(* PLC project 117_1_V0.5.project, CODESYS CODESYS V3.5 SP17 Patch 3 *)
(* stored: creationDateTime 1970-01-01T00:00:00, modificationDateTime 2026-03-26T18:14:32.4070562 *)

FUNCTION_BLOCK TestingForces_150321
  VAR_INPUT
    A : E_A;
  END_VAR
  VAR_OUTPUT
    Fstab : UDINT;
    Fset : UDINT;
    Fsp : UDINT;
    F_su_lower_level : UDINT;
    F_su_upper_level : UDINT;
  END_VAR

            CASE A OF
	
	A60:
				Fstab				:= 50;
				Fset				:= 720;
				Fsp					:= 1575;	
				
 				F_su_lower_level	:= 2363;		
				F_su_upper_level	:= 3150;
	
	A80: 
				Fstab				:= 50;
				Fset				:= 840; 
				Fsp					:= 1838;
				
				F_su_lower_level	:= 2756;
				F_su_upper_level	:= 3675;

	A100:
				Fstab				:= 50;
				Fset				:= 1024;
				Fsp					:= 2240;
				
				F_su_lower_level	:= 3360;
				F_su_upper_level	:= 4480;
						
END_CASE
          
END_FUNCTION_BLOCK
